TYPE WcStateBase_A2171C4E :
STRUCT
END_STRUCT
END_TYPE

(* stored: Version 1.1.0.1, ProductVersion 3.1.4024.9
   DUT WcStateBase_A2171C4E: Id {cdf20fc1-2245-055f-3587-cbe8a6677039} *)
